Fanuc KAREL source: kb00003.KL

-- PROVISIONAL review KL for V1013-1; original PC SHA256 bd23c1971cc715c9a96160d02604e26af708c8c357b3d1ea05a7e313a2c1e927
-- Incomplete behavior may be omitted. Consult companion uncertainty JSON. Do not deploy.
PROGRAM KB00003
%NOLOCKGROUP
VAR
  P1 : REAL
  RESULT : REAL
BEGIN
  -- UNRESOLVED_PC offsets 5-16; opcodes 2E,23
  -- UNRESOLVED_PC offsets 21-36; opcodes 27,22,76,23
  -- UNRESOLVED_PC offsets 41-45; opcodes 7F
END KB00003
